// TIA Portal V20 export
VAR_GLOBAL   // PLC tag table "BW_Inputs"
   AI_LifeFlag AT %IW500 : Int;
   DI_JobDone AT %I502.0 : Bool;
   DI_LockShuttle AT %I504.0 : Bool;
   AI_DataSend AT %IW506 : Int;
   AI_DataReceive AT %IW508 : Int;
   DI_NoEmergencyStopAtBwLoader AT %I510.0 : Bool;
   DI_SafetyDoorsClosedAtBwLoader AT %I512.0 : Bool;
   AI_BwInErrorState AT %IW514 : Int;
   DI_UndrilledPartControl AT %I516.0 : Bool;
   DI_DrilledPartControl AT %I518.0 : Bool;
   DI_BackwallControl AT %I520.0 : Bool;
   DI_BwLoaderInSafePos AT %I522.0 : Bool;
   DI_SemiAutoValid AT %I562.0 : Bool;
END_VAR
